TYPE ST_EVENT :
STRUCT
	
	bImmediateFault						: BOOL;
	bCycleStopFault						: BOOL;
	bCycleStopRequest					: BOOL;
	bMessage							: BOOL;
	
	bAssignedID							: DINT;
	
	bEventFlag							: BOOL;
	bEventTimer							: TON;
	bEventText							: STRING(255);
	bEventTextHMI						: STRING(255);
	sSolution							: STRING(255);
	bActive								: BOOL;

END_STRUCT
END_TYPE

(* stored: Version 1.1.0.1, ProductVersion 3.1.4024.13
   DUT ST_EVENT: Id {aa8240d2-f153-4b6d-8ba3-f39478af10c7} *)
